{attribute 'qualified_only'}
TYPE E_RobotAddress :
(
	Undefined := 0,
	Address01,
	Address02,
	Address03,
	Address04,
	Address05,
	Address06
);
END_TYPE

(* stored: Version 1.1.0.1, ProductVersion 3.1.4024.13
   DUT E_RobotAddress: Id {dd21978f-5367-40b1-8dc9-b3a53edaa8c5} *)
